(* IEC 61131-3 sources: verifaps-lib/util/src/testFixtures/resources/edu/kit/iti/formal/automation/st/programs, 14 files *)

(* ---- type_ampel.st ---- *)
TYPE
    (*  Rot hat den Initialwert 0, Gelb 1, Gruen 10 *)
    AMPEL: (Rot, Gelb, Gruen := 10);
END_TYPE

(* ---- interface.st ---- *)
INTERFACE abc

  METHOD PUBLIC foo
    VAR_INPUT
      i : INT;
    END_VAR
  END_METHOD

END_INTERFACE

INTERFACE empty
END_INTERFACE

INTERFACE intf EXTENDS abc, empty
  METHOD com
    VAR_INPUT
      s : STRING;
    END_VAR
  END_METHOD
END_INTERFACE

INTERFACE ROOM
  METHOD DAYTIME
  END_METHOD
  METHOD NIGHTTIME
  END_METHOD
END_INTERFACE

(* ---- func_sel.st ---- *)
(* Selection function, typical built-in
 *
 *)
FUNCTION SEL : BOOL
    VAR_INPUT
        a : BOOL;
        b : BOOL;
        c : BOOL;
    END_VAR
    IF a THEN SEL := b; ELSE SEL := c; END_IF
END_FUNCTION

(* ---- arrays.st ---- *)
CLASS A
  VAR
    a : ARRAY [0..7] OF INT := [7(1)];
    b : ARRAY [0..2] OF STRING := ["a", "b", "c"];
  END_VAR
END_CLASS

(* ---- assignment_attempt.st ---- *)
INTERFACE ITF1
END_INTERFACE

INTERFACE ITF2
END_INTERFACE

INTERFACE ITF3
END_INTERFACE

CLASS C IMPLEMENTS ITF1, ITF2
END_CLASS

PROGRAM A
  VAR
    inst: C;
    interf1: ITF1;
    interf2: ITF2;
    interf3: ITF3;
  END_VAR

interf1 := inst;
interf2 ?= interf1;
interf3 ?= interf1;

END_PROGRAM

(* ---- circle.st ---- *)
CLASS ABSTRACT GEOMETRY
END_CLASS

CLASS CIRCLE EXTENDS GEOMETRY

METHOD PUBLIC PI: LREAL
  PI := 3.1415;
END_METHOD

METHOD PUBLIC CF: LREAL
  VAR_INPUT DIAMETER: LREAL; END_VAR
  CF := THIS.PI() + 3;
  CF := THIS.PI() * DIAMETER;
END_METHOD
END_CLASS

CLASS FINAL CIRCLE2 EXTENDS CIRCLE

METHOD PUBLIC OVERRIDE PI: LREAL
  PI := 3.1415926;
END_METHOD
END_CLASS

PROGRAM TEST
VAR
  CIR1: CIRCLE;
  CIR2: CIRCLE2;
  CUMF1: LREAL;
  CUMF2: LREAL;
  DYNAMIC: BOOL;
END_VAR

CUMF1 := CIR1.CF(1.0);
CUMF2 := CIR2.CF(1.0);
DYNAMIC := CUMF1 <> CUMF2;

END_PROGRAM

(* ---- class_initialization.st ---- *)
CLASS ID_Card
  VAR
    id : INT;
  END_VAR
END_CLASS

CLASS Student
  VAR
    id_card : ID_Card;
    name : STRING;
  END_VAR
END_CLASS

CLASS Verifier
  METHOD verify : BOOL
    VAR_INPUT
      id_card : ID_Card;
    END_VAR

    (* Super-secure verification *)
    IF (id_card.id > 9) THEN
      verify := TRUE;
    ELSE
      verify := FALSE;
    END_IF
  END_METHOD
END_CLASS

PROGRAM MyProgram
  VAR
    student_id_card : ID_Card := (id := 42);
    student : Student := (id := (id:=42), name := "Toby");
    fake_student : Student := (id_card := null, name := "Victor");
    verif : Verifier;
  END_VAR

  verif.verify(student.id_card); // TRUE
  verif.verify(fake_student.id_card); // FALSE
END_PROGRAM

(* ---- classes.st ---- *)
INTERFACE ROOM
  METHOD DAYTIME END_METHOD

  METHOD NIGHTTIME END_METHOD
END_INTERFACE

FUNCTION_BLOCK ROOM_CTRL

    VAR_EXTERNAL
      DAYTIME : DATE; // global time definition
    END_VAR

    VAR_INPUT
      RM : ROOM;
    END_VAR

    IF (RM = NULL) THEN // always test on valid reference!
        RETURN;
    END_IF

    IF DAYTIME >= TOD#20:15 OR DAYTIME <= TOD#6:00 THEN
        RM.NIGHTTIME();
    ELSE
        RM.DAYTIME();
    END_IF
END_FUNCTION_BLOCK

FUNCTION_BLOCK LIGHTROOM IMPLEMENTS ROOM
VAR
LIGHT : BOOL;
END_VAR
METHOD PUBLIC DAYTIME : VOID
LIGHT := FALSE;
END_METHOD
METHOD PUBLIC NIGHTTIME : VOID
LIGHT := TRUE;
END_METHOD
END_FUNCTION_BLOCK

FUNCTION_BLOCK LIGHT2ROOM EXTENDS LIGHTROOM
VAR
  LIGHT2 : BOOL;
END_VAR

METHOD PUBLIC DAYTIME : VOID
  SUPER.DAYTIME ();
  // call of parent implementation
  LIGHT2 := FALSE;
END_METHOD

METHOD PUBLIC NIGHTTIME : VOID
  SUPER.NIGHTTIME ();
  // call of parent implementation
  LIGHT2 := TRUE;
END_METHOD

END_FUNCTION_BLOCK

(* ---- Crane.st ---- *)
TYPE
    Crane_states_t : (Crane_Go_Up , Crane_Init , Crane_Init_2 , Crane_Lift_At_Stamp , Crane_Lift_Conveyor , Crane_Lift_Conveyor_Black , Crane_Lift_Magazin , Crane_Lift_Magazin_Metallic , Crane_Lift_NOT_Metallic_Black , Crane_Lower , Crane_On_Conveyor , Crane_On_Conveyor_Metallic , Crane_On_Conveyor_Not_Metallica_Black , Crane_On_Stamp_Metallic , Crane_On_Stamp_Stop_Black , Crane_Turn_Left_Back_To_Stamp , Crane_Turn_Left_From_Stamp , Crane_Turn_Left_Metallic , Crane_Turn_Left_NOT_Metallic , Crane_Turn_Left_NOT_Metallic_Black , Init , Interstep , Interstep_2 , Last_Workpiece_At_Stamp , Lower_Crane , Magazin_Stop , Magazin_Stop_Black , No_Workpiece_ready , Reset_interconnect , Start_Crane , Step0 , Suck_At_Stamp , TimeDelay , Turn_Right , Turn_Right_Black , pause , release , release_Black , release_Workpiece);
END_TYPE

FUNCTION_BLOCK TON

VAR_INPUT
    IN : BOOL;
    PT : USINT;
END_VAR

VAR_OUTPUT
    Q  : BOOL;
    ET : USINT;
END_VAR

IF IN THEN
    Q:= ET = USINT#0;
    IF ET > USINT#0 THEN
        ET := ET - USINT#1;
    ELSE
        ET := USINT#0;
    END_IF
ELSE
    Q  := FALSE;
    ET := PT;
END_IF

END_FUNCTION_BLOCK

PROGRAM Crane
    VAR  CranTurnClockwise : BOOL; END_VAR
    VAR_INPUT  CraneDown : BOOL; END_VAR
    VAR_OUTPUT  CraneLower : BOOL; END_VAR
    VAR_INPUT  CraneOnConveyor : BOOL; END_VAR
    VAR_INPUT  CraneOnMagazin : BOOL; END_VAR
    VAR_INPUT  CranePositionStamp : BOOL; END_VAR
    VAR_INPUT  CraneSucked : BOOL; END_VAR
    VAR_OUTPUT  CraneTurnClockwise : BOOL; END_VAR
    VAR_OUTPUT  CraneTurnCounterclockwise : BOOL; END_VAR
    VAR_INPUT  CraneUp : BOOL; END_VAR
    VAR  Duration1 : TIME := TIME#1.0s500.0ms; END_VAR
    VAR_INPUT  MagazinCapacitiveSensor : BOOL; END_VAR
    VAR_OUTPUT  MagazinSlider : BOOL; END_VAR
    VAR_OUTPUT  MagazinVacuumOff : BOOL; END_VAR
    VAR_OUTPUT  MagazinVacuumOn : BOOL; END_VAR
    VAR  SFCInit : BOOL; END_VAR
    VAR_INPUT  SFCReset : BOOL; END_VAR
    VAR_INPUT  SliderMovedOut : BOOL; END_VAR
    VAR_INPUT  SliderNotMovedOut : BOOL; END_VAR
    VAR_INPUT  StampLowered : BOOL; END_VAR
    VAR_INPUT  StampSliderFilled : BOOL; END_VAR
    VAR_INPUT  StartButtonMagazin : BOOL; END_VAR
    VAR_OUTPUT  StartCommandCrane : BOOL; END_VAR
    VAR_INPUT  StartVar : BOOL; END_VAR
    VAR  TimeDelay_Timer : TON; END_VAR
    VAR  TimeDelay_Timer_Duration : TIME := TIME#50.0ms; END_VAR
    VAR  TimeDelay_Timer_interconnect : BOOL; END_VAR
    VAR  Timer1 : TON; END_VAR
    VAR_INPUT  WorkpieceReady : BOOL; END_VAR
    VAR  _state : Crane_states_t; END_VAR
    VAR  _transit : BOOL; END_VAR
    VAR  actualtime1 : TIME; END_VAR
    VAR  interconnect : BOOL; END_VAR
    VAR  interconnectCraneStartCommand : BOOL; END_VAR

    CASE _state OF
        Crane_states_t#Crane_Go_Up:
            _transit := FALSE;
            CraneLower := FALSE;
            IF (CraneUp AND (MagazinCapacitiveSensor OR NOT WorkpieceReady)) THEN
                _transit := TRUE;
                _state := Crane_states_t#pause;
            ELSEIF ((CraneUp AND NOT MagazinCapacitiveSensor) AND WorkpieceReady) THEN
                _transit := TRUE;
                _state := Crane_states_t#Turn_Right_Black;
            END_IF

        Crane_states_t#Crane_Init:
            _transit := FALSE;
            CraneLower := TRUE;
            interconnectCraneStartCommand := FALSE;
            IF CraneDown THEN
                _transit := TRUE;
                _state := Crane_states_t#Crane_Init_2;
            END_IF

        Crane_states_t#Crane_Init_2:
            _transit := FALSE;
            CraneLower := FALSE;
            IF CraneUp THEN
                _transit := TRUE;
                _state := Crane_states_t#Interstep;
            END_IF

        Crane_states_t#Crane_Lift_At_Stamp:
            _transit := FALSE;
            CraneLower := FALSE;
            IF CraneUp THEN
                _transit := TRUE;
                _state := Crane_states_t#Crane_Turn_Left_From_Stamp;
            END_IF

        Crane_states_t#Crane_Lift_Conveyor:
            _transit := FALSE;
            CraneLower := FALSE;
            IF TRUE THEN
                _transit := TRUE;
                _state := Crane_states_t#Interstep;
            END_IF

        Crane_states_t#Crane_Lift_Conveyor_Black:
            _transit := FALSE;
            CraneLower := FALSE;
            IF CraneUp THEN
                _transit := TRUE;
                _state := Crane_states_t#Crane_Turn_Left_Back_To_Stamp;
            END_IF

        Crane_states_t#Crane_Lift_Magazin:
            _transit := FALSE;
            CraneLower := FALSE;
            IF CraneUp THEN
                _transit := TRUE;
                _state := Crane_states_t#Crane_Turn_Left_NOT_Metallic;
            END_IF

        Crane_states_t#Crane_Lift_Magazin_Metallic:
            _transit := FALSE;
            CraneLower := FALSE;
            IF CraneUp THEN
                _transit := TRUE;
                _state := Crane_states_t#Crane_Turn_Left_Metallic;
            END_IF

        Crane_states_t#Crane_Lift_NOT_Metallic_Black:
            _transit := FALSE;
            CraneLower := FALSE;
            IF CraneUp THEN
                _transit := TRUE;
                _state := Crane_states_t#Crane_Turn_Left_NOT_Metallic_Black;
            END_IF

        Crane_states_t#Crane_Lower:
            _transit := FALSE;
            MagazinVacuumOn := TRUE;
            MagazinVacuumOff := FALSE;
            CraneLower := TRUE;
            IF CraneSucked THEN
                _transit := TRUE;
                _state := Crane_states_t#Step0;
            END_IF

        Crane_states_t#Crane_On_Conveyor:
            _transit := FALSE;
            CraneTurnCounterclockwise := FALSE;
            CraneTurnClockwise := FALSE;
            CraneLower := TRUE;
            IF CraneDown THEN
                _transit := TRUE;
                _state := Crane_states_t#release;
            END_IF

        Crane_states_t#Crane_On_Conveyor_Metallic:
            _transit := FALSE;
            CraneTurnCounterclockwise := FALSE;
            CraneTurnClockwise := FALSE;
            CraneLower := TRUE;
            IF CraneDown THEN
                _transit := TRUE;
                _state := Crane_states_t#release;
            END_IF

        Crane_states_t#Crane_On_Conveyor_Not_Metallica_Black:
            _transit := FALSE;
            CraneTurnCounterclockwise := FALSE;
            CraneTurnClockwise := FALSE;
            CraneLower := TRUE;
            IF CraneDown THEN
                _transit := TRUE;
                _state := Crane_states_t#release_Black;
            END_IF

        Crane_states_t#Crane_On_Stamp_Metallic:
            _transit := FALSE;
            CraneTurnCounterclockwise := FALSE;
            CraneTurnClockwise := FALSE;
            CraneLower := TRUE;
            IF CraneDown THEN
                _transit := TRUE;
                _state := Crane_states_t#release_Workpiece;
            END_IF

        Crane_states_t#Crane_On_Stamp_Stop_Black:
            _transit := FALSE;
            CraneTurnClockwise := FALSE;
            CraneTurnCounterclockwise := FALSE;
            IF TRUE THEN
                _transit := TRUE;
                _state := Crane_states_t#Reset_interconnect;
            END_IF

        Crane_states_t#Crane_Turn_Left_Back_To_Stamp:
            _transit := FALSE;
            CraneTurnCounterclockwise := TRUE;
            CraneTurnClockwise := FALSE;
            IF CranePositionStamp THEN
                _transit := TRUE;
                _state := Crane_states_t#Crane_On_Stamp_Stop_Black;
            END_IF

        Crane_states_t#Crane_Turn_Left_From_Stamp:
            _transit := FALSE;
            CraneTurnClockwise := TRUE;
            CraneTurnCounterclockwise := FALSE;
            IF CraneOnConveyor THEN
                _transit := TRUE;
                _state := Crane_states_t#Crane_On_Conveyor_Metallic;
            END_IF

        Crane_states_t#Crane_Turn_Left_Metallic:
            _transit := FALSE;
            CraneTurnCounterclockwise := TRUE;
            CraneTurnClockwise := FALSE;
            IF CranePositionStamp THEN
                _transit := TRUE;
                _state := Crane_states_t#Crane_On_Stamp_Metallic;
            END_IF

        Crane_states_t#Crane_Turn_Left_NOT_Metallic:
            _transit := FALSE;
            CraneTurnCounterclockwise := TRUE;
            CraneTurnClockwise := FALSE;
            IF CraneOnConveyor THEN
                _transit := TRUE;
                _state := Crane_states_t#Crane_On_Conveyor;
            END_IF

        Crane_states_t#Crane_Turn_Left_NOT_Metallic_Black:
            _transit := FALSE;
            CraneTurnCounterclockwise := TRUE;
            CraneTurnClockwise := FALSE;
            IF CraneOnConveyor THEN
                _transit := TRUE;
                _state := Crane_states_t#Crane_On_Conveyor_Not_Metallica_Black;
            END_IF

        Crane_states_t#Init:
            _transit := FALSE;
            IF TRUE THEN
                _transit := TRUE;
                _state := Crane_states_t#Start_Crane;
            END_IF

        Crane_states_t#Interstep:
            _transit := FALSE;
            StartCommandCrane := TRUE;
            IF StartVar THEN
                _transit := TRUE;
                _state := Crane_states_t#Interstep_2;
            END_IF

        Crane_states_t#Interstep_2:
            _transit := FALSE;
            IF SliderMovedOut THEN
                _transit := TRUE;
                _state := Crane_states_t#TimeDelay;
            END_IF

        Crane_states_t#Last_Workpiece_At_Stamp:
            _transit := FALSE;
            IF TRUE THEN
                _transit := TRUE;
                _state := Crane_states_t#pause;
            END_IF

        Crane_states_t#Lower_Crane:
            _transit := FALSE;
            CraneLower := TRUE;
            IF CraneDown THEN
                _transit := TRUE;
                _state := Crane_states_t#Suck_At_Stamp;
            END_IF

        Crane_states_t#Magazin_Stop:
            _transit := FALSE;
            CraneTurnClockwise := FALSE;
            CraneTurnCounterclockwise := FALSE;
            IF (NOT WorkpieceReady AND NOT StampSliderFilled) THEN
                _transit := TRUE;
                _state := Crane_states_t#No_Workpiece_ready;
            ELSEIF WorkpieceReady THEN
                _transit := TRUE;
                _state := Crane_states_t#Crane_Lower;
            ELSEIF (NOT WorkpieceReady AND StampSliderFilled) THEN
                _transit := TRUE;
                _state := Crane_states_t#Last_Workpiece_At_Stamp;
            END_IF

        Crane_states_t#Magazin_Stop_Black:
            _transit := FALSE;
            CraneTurnClockwise := FALSE;
            CraneTurnCounterclockwise := FALSE;
            MagazinVacuumOn := TRUE;
            MagazinVacuumOff := FALSE;
            CraneLower := TRUE;
            IF CraneSucked THEN
                _transit := TRUE;
                _state := Crane_states_t#Crane_Lift_NOT_Metallic_Black;
            END_IF

        Crane_states_t#No_Workpiece_ready:
            _transit := FALSE;
            IF TRUE THEN
                _transit := TRUE;
                _state := Crane_states_t#Start_Crane;
            END_IF

        Crane_states_t#Reset_interconnect:
            _transit := FALSE;
            interconnect := FALSE;
            Timer1(IN := FALSE, PT := TIME#1.0ms);
            IF SliderMovedOut THEN
                _transit := TRUE;
                _state := Crane_states_t#Lower_Crane;
            END_IF

        Crane_states_t#Start_Crane:
            _transit := FALSE;
            CraneLower := FALSE;
            MagazinVacuumOff := TRUE;
            MagazinVacuumOn := FALSE;
            CraneTurnCounterclockwise := FALSE;
            CraneTurnClockwise := FALSE;
            StartVar := FALSE;
            StartCommandCrane := FALSE;
            IF (StartButtonMagazin = TRUE) THEN
                interconnectCraneStartCommand := TRUE;
            END_IF
            IF interconnectCraneStartCommand THEN
                _transit := TRUE;
                _state := Crane_states_t#Crane_Init;
            END_IF

        Crane_states_t#Step0:
            _transit := FALSE;
            IF NOT MagazinCapacitiveSensor THEN
                _transit := TRUE;
                _state := Crane_states_t#Crane_Lift_Magazin;
            ELSEIF MagazinCapacitiveSensor THEN
                _transit := TRUE;
                _state := Crane_states_t#Crane_Lift_Magazin_Metallic;
            END_IF

        Crane_states_t#Suck_At_Stamp:
            _transit := FALSE;
            MagazinVacuumOn := TRUE;
            MagazinVacuumOff := FALSE;
            IF CraneSucked THEN
                _transit := TRUE;
                _state := Crane_states_t#Crane_Lift_At_Stamp;
            END_IF

        Crane_states_t#TimeDelay:
            _transit := FALSE;
            TimeDelay_Timer(IN := TRUE, PT := TimeDelay_Timer_Duration);
            TimeDelay_Timer_interconnect := TimeDelay_Timer.Q;
            IF TimeDelay_Timer_interconnect THEN
                _transit := TRUE;
                _state := Crane_states_t#Turn_Right;
            END_IF

        Crane_states_t#Turn_Right:
            _transit := FALSE;
            CraneTurnClockwise := TRUE;
            CraneTurnCounterclockwise := FALSE;
            IF CraneOnMagazin THEN
                _transit := TRUE;
                _state := Crane_states_t#Magazin_Stop;
            END_IF

        Crane_states_t#Turn_Right_Black:
            _transit := FALSE;
            CraneTurnClockwise := TRUE;
            CraneTurnCounterclockwise := FALSE;
            IF CraneOnMagazin THEN
                _transit := TRUE;
                _state := Crane_states_t#Magazin_Stop_Black;
            END_IF

        Crane_states_t#pause:
            _transit := FALSE;
            Timer1(IN := CraneUp, PT := Duration1);
            interconnect := Timer1.Q;
            IF interconnect THEN
                _transit := TRUE;
                _state := Crane_states_t#Reset_interconnect;
            END_IF

        Crane_states_t#release:
            _transit := FALSE;
            MagazinVacuumOff := TRUE;
            MagazinVacuumOn := FALSE;
            IF TRUE THEN
                _transit := TRUE;
                _state := Crane_states_t#Crane_Lift_Conveyor;
            END_IF

        Crane_states_t#release_Black:
            _transit := FALSE;
            MagazinVacuumOn := FALSE;
            MagazinVacuumOff := TRUE;
            IF TRUE THEN
                _transit := TRUE;
                _state := Crane_states_t#Crane_Lift_Conveyor_Black;
            END_IF

        Crane_states_t#release_Workpiece:
            _transit := FALSE;
            MagazinVacuumOff := TRUE;
            MagazinVacuumOn := FALSE;
            IF TRUE THEN
                _transit := TRUE;
                _state := Crane_states_t#Crane_Go_Up;
            END_IF

            END_CASE
END_PROGRAM

(* ---- effective_subtypes.st ---- *)
INTERFACE ITF END_INTERFACE
CLASS A IMPLEMENTS ITF END_CLASS
CLASS B EXTENDS A END_CLASS
CLASS C EXTENDS A END_CLASS

PROGRAM MY_PROGRAM
  VAR
    a : A;
    b : B;
    i : ITF;
    r : REF_TO A;
  END_VAR

    VAR_INPUT
      switch : BOOL;
    END_VAR

  IF (switch) THEN
    i := a;
    r := REF(a);
  ELSE
    i := b;
    r := REF(b);
  END_IF
END_PROGRAM

(* ---- instance_hierarchy.st ---- *)
CLASS C

  VAR
    ID : INT;
  END_VAR

END_CLASS

CLASS B

  VAR
    MY_C : C := (ID := 42);
  END_VAR

END_CLASS

CLASS A

  VAR
    B1 : B;
    B2 : B;
  END_VAR

END_CLASS

PROGRAM MY_PROGRAM
  VAR
    MY_A : A;
    MY_B : B;
    MY_C : C;
  END_VAR

END_PROGRAM

(* ---- pass_by_ref.st ---- *)
CLASS C
  VAR PUBLIC
    a : INT := 42;
    b : INT := 33;
  END_VAR
END_CLASS

CLASS Util
  METHOD PUBLIC modify_c
    VAR_INPUT
      c : REF_TO C;
    END_VAR

    c^.a := c^.a + c^.b;
  END_METHOD
END_CLASS

PROGRAM A
  VAR
    c1 : C;
    c2 : C := (a := 10, b := 10);
    u : Util;
  END_VAR

  u.modify_c(c := c1);  // c1.a == 75
  u.modify_c(c := c2);  // c1.b == 20
  u.modify_c(c := c2);  // c1.b == 30
END_PROGRAM

(* ---- references.st ---- *)
INTERFACE ITF1
  METHOD func : INT
  END_METHOD
END_INTERFACE

INTERFACE ITF2
END_INTERFACE

INTERFACE ITF3
END_INTERFACE

CLASS ClBase IMPLEMENTS ITF1, ITF2
  VAR
    x : INT;
  END_VAR

  METHOD func : INT
    func := 42;
  END_METHOD
END_CLASS

CLASS ClDerived EXTENDS ClBase
  METHOD func : INT
    func := 24;
  END_METHOD
END_CLASS

PROGRAM A
  VAR
    instBase : ClBase;
    instDerived: ClDerived;
    rinstBase1, rinstBase2: REF_TO ClBase;
    rinstDerived1, rinstDerived2: REF_TO ClDerived;
    rinstDerived3, rinstDerived4: REF_TO ClDerived;
    interf1: ITF1;
    interf2: ITF2;
    interf3: ITF3;
  END_VAR

rinstBase1:= REF(instBase); // rinstbase1 references base class
rinstBase2:= REF(instDerived); // rinstbase2 references derived class

rinstDerived1 ?= rinstBase1; // rinstDerived1 == NULL
rinstDerived2 ?= rinstBase2; // rinstDerived2 will contain a valid
                             // reference to instDerived
interf1:= instBase;    // interf1 is a reference to base class
interf2:= instDerived; // interf2 is a reference to derived class

rinstDerived3 ?= interf1; // rinstDerived3 == NULL
rinstDerived4 ?= interf2; // rinstDerived4 will contain a valid
                          // reference to instDerived

rinstBase1:= REF(instBase); // rinstbase1 references base class
rinstBase2:= REF(instDerived); // rinstbase2 references derived class

rinstBase1^.x := interf1.func();  // 42
rinstBase2^.x := interf2.func();  // 24

END_PROGRAM

(* ---- program_with_actions.st ---- *)
PROGRAM abc
    VAR
        s : INT;
    END_VAR

    VAR_INPUT
        i : INT;
    END_VAR

    VAR_OUTPUT
        o : INT;
    END_VAR

    ACTION up
        s := (s + i);
    END_ACTION
    ACTION down
        s := (s - i);
    END_ACTION

    IF (i < INT#0) THEN
        down();
    ELSE
        up();
    END_IF
    o := s;
END_PROGRAM
